// Mitsubishi GX Works2 project: a07   PLC: Q02/Q02H

PROGRAM MAIN
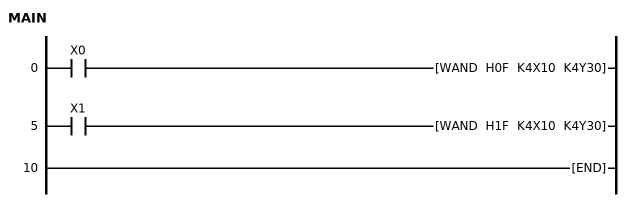
0     LD      X0
      WAND    H0F K4X10 K4Y30
5     LD      X1
      WAND    H1F K4X10 K4Y30
10    END
END_PROGRAM
